{attribute 'no_check'}
//Generic Unit 
FUNCTION_BLOCK Statemodel_Unit implements I_Statemodel_Unit
VAR_OUTPUT CONSTANT
END_VAR             										
VAR_INPUT
{attribute 'TcHmiSymbol.AddSymbol'}                      										
	Unit																:	Statemodel;		
END_VAR             										
VAR_OUTPUT          										
END_VAR             	
VAR                 	
(* Local variables ************************************************************)

(* Trigger *****************************************************************)

(* Timer ******************************************************************)

(* Fcuntion blocks ***************************************************************)

(* Dummys **********************************************************)

END_VAR

	(* Generic unit incl. state model										V1.0		*)
	(************************************************************************************)

(* work local sub ****************************************)
	Unit();
	IF Unit.RT_StateChanged THEN stateChanged(unit.Mode, Unit.State); END_IF
	
(* call methods ********************************************)
	CASE Unit.state OF
	eSTATE.STARTUP			:	startup();
	eSTATE.IDLE				: 	idle();
	eSTATE.STARTING			:	starting();		
	eSTATE.STARTED			: 	started();	
	eSTATE.EXECUTE			:	executing();
	eSTATE.COMPLETING		:	completing();
	eSTATE.COMPLETE			: 	complete();
	eSTATE.ABORTING			:	aborting();
	eSTATE.ABORTED			:  	aborted();
	eSTATE.CLEARING			:	clearing();
	eSTATE.STOPPING			:	stopping();
	eSTATE.STOPPED			: 	stopped();
	eSTATE.RESETTING		:	resetting();
	ELSE
		;
	END_CASE

(*********************************************************)

METHOD PROTECTED aborted : BOOL
VAR_INPUT
END_VAR
Aborted														:= unit.InAborted;
END_METHOD

METHOD PROTECTED aborting : BOOL
VAR_INPUT
END_VAR
Unit.StateComplete();
Aborting													:= Unit.InAborting;
END_METHOD

METHOD PROTECTED clearing : Bool
VAR_INPUT
END_VAR
Unit.StateComplete();
Clearing													:= Unit.InClearing;
END_METHOD

METHOD PROTECTED complete : Bool
VAR_INPUT
END_VAR
Complete														:= unit.InComplete;
END_METHOD

METHOD PROTECTED completing : BOOL
VAR_INPUT
END_VAR
Unit.StateComplete();
Completing													:= Unit.InCompleting;
END_METHOD

METHOD PROTECTED executing : booL
VAR_INPUT
END_VAR
Executing 												:= Unit.InExecute;
END_METHOD

METHOD FB_exit : BOOL
VAR_INPUT
	bInCopyCode : BOOL; // if TRUE, the exit method is called for exiting an instance that is copied afterwards (online change).
END_VAR
FB_EXit															:= TRUE;
END_METHOD

METHOD FB_init : BOOL
VAR_INPUT
	bInitRetains : BOOL; // if TRUE, the retain variables are initialized (warm start / cold start)
	bInCopyCode : BOOL;  // if TRUE, the instance afterwards gets moved into the copy code (online change)
END_VAR
(* Example 
	Unit.pSubRemoteData[1]												:= ADR(Infeed.unit.RemoteData);
	Unit.pSubRemoteData[2]												:= ADR(Support_1.unit.RemoteData);
	Unit.pSubRemoteData[3]												:= ADR(Support_2.RemoteData);	
	Unit.pSubRemoteData[4]												:= ADR(Transport.unit.RemoteData);
	Unit.pSubRemoteData[5]												:= ADR(Outfeed.unit.RemoteData);
*)
FB_init														:= TRUE;
END_METHOD

METHOD FB_reinit : BOOL
VAR_INPUT
END_VAR
FB_reinit											:= TRUE;
END_METHOD

METHOD PROTECTED idle : Bool
VAR_INPUT
END_VAR
Idle														:= unit.InIdle;
END_METHOD

METHOD PROTECTED Resetting : Bool
VAR_INPUT
END_VAR
Unit.StateComplete();
Resetting													:= Unit.InResetting;
END_METHOD

{attribute 'monitoring' := 'call'}
PROPERTY public rUnit : REFERENCE TO Statemodel
GET
rUnit REF= Unit;
END_GET
END_PROPERTY

METHOD PROTECTED started : Bool
VAR_INPUT
END_VAR
Started													:= Unit.InStarted;
END_METHOD

METHOD PROTECTED starting : Bool
VAR_INPUT
END_VAR
Unit.StateComplete();
Starting													:= Unit.InStarting;
END_METHOD

METHOD PROTECTED startup : Bool
VAR_INPUT
END_VAR
Unit.StateComplete();
Startup													:= Unit.InStartup;
END_METHOD

METHOD PROTECTED stateChanged : BOOL 
VAR_INPUT
	mode											:	eMODE;
	state											:	eSTATE;
END_VAR
END_METHOD

METHOD PROTECTED stopped : Bool
VAR_INPUT
END_VAR
Stopped														:= unit.InStopped;
END_METHOD

METHOD PROTECTED stopping : Bool
VAR_INPUT
END_VAR
Unit.StateComplete();
Stopping													:= Unit.InStopping;
END_METHOD

END_FUNCTION_BLOCK

(* stored: Version 1.1.0.1, ProductVersion 3.1.4024.13
   POU Statemodel_Unit: Id {ebc3bf14-2e73-4603-a8d5-3e529b9caa55}, SpecialFunc None
   Method aborted: Id {82094b5b-6c33-4c21-8f74-3ef83fdda4b0}
   Method aborting: Id {e8d115e6-dacd-49ec-aaf4-ce4634199a7e}
   Method clearing: Id {b645cd56-0f2c-40b6-9f98-6e3021eddf44}
   Method complete: Id {f49be510-fde6-4b8e-8472-ddd3432d34ad}
   Method completing: Id {0f6bc1fe-5d74-45dc-ae55-bd8fc050dd90}
   Method executing: Id {efff44cc-82de-4521-a0c8-89a79699f984}
   Method FB_exit: Id {df18465b-7f5d-45ef-a504-49d789b5e3ae}
   Method FB_init: Id {9e160fa4-7328-4996-8c5d-105b3eb3659e}
   Method FB_reinit: Id {793f5187-7f65-4e6f-9205-335d5e3901d8}
   Method idle: Id {be30ccff-9ac6-4518-af4e-c31398a52757}
   Method resetting: Id {07d90871-ac01-4b0e-a034-21db6a2d45f2}
   Property rUnit: Id {deb3908d-d327-41b8-afea-a807f10a2d4d}
   Get Get: Id {6d48cdd0-6fc5-4986-98f2-40c49cd2e3c3}
   Method started: Id {2f6dcd2f-f0fb-475f-8015-19a506e88f5b}
   Method starting: Id {f4e5aa13-f5ca-4240-b851-6eb873bd50d1}
   Method startup: Id {d2518eb1-0622-42af-9c21-6e180208979e}
   Method stateChanged: Id {6665c611-5b14-4afd-9cb8-4b1ba0090389}
   Method stopped: Id {0d21fbd5-68a0-426c-98fc-91a6b3e502a4}
   Method stopping: Id {cd9dce3e-ab88-4ce7-a46d-aedd1f84bb60} *)
